TYPE E_CircuitBreakerPosition :
(
    UNDEFINED := 0,     // Belirsiz durum
    OFF := 1,           // OFF pozisyonu
    ON := 2,            // ON pozisyonu
    TRIPPED := 3        // TRIP pozisyonu
);
END_TYPE

(* stored: Version 1.1.0.1, ProductVersion 3.1.4024.15
   EnumerationTextList E_CircuitBreakerPosition: Id {0dfd97cf-05b2-4131-8ef5-a8495b974a00} *)
